# EPICS StreamDevice protocol: protocols/sfp.proto
Terminator = CR LF;
ExtraInput = Ignore;

#Temp:  31.28 C
#VCC:   3.26 V
#Tx Bias:1492.50 uA
#Tx Power: 429.90 uW
#Rx Pwr: 454.10 uW

getTemp {
	in "\_Temp:\_%f C";
}

getVCC {
	in "\_VCC:\_%f V"
}

getRxPwr {
	in "\_Rx Pwr:\_%f uW";
}

getTxPwr {
	in "\_Tx Power:\_%f uW"
}

getTxBias {
	in "\_Tx Bias:%f uA";
}
